RoboDK station: New Station (1).rdk

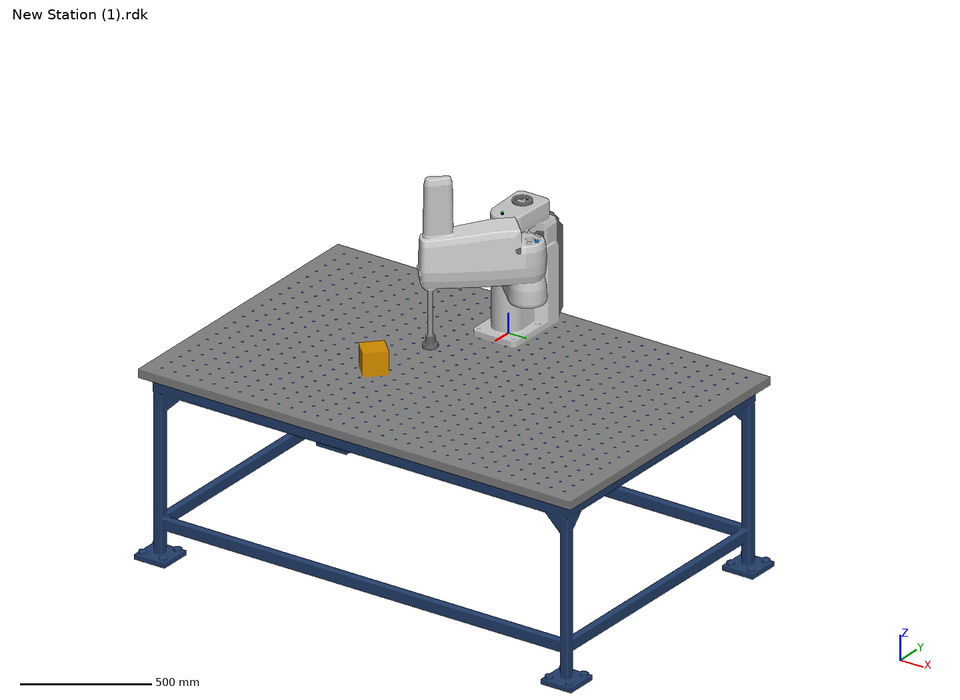
[picture v0: the station drawn from its stored meshes, robots at their saved joint values, targets as dots, program paths as lines]
Station New Station (1) (saved by RoboDK 5.3.2). Poses are relative to the parent item; angles as X-Y-Z fixed-axis rotations.
  - frame Adept Cobra s800 Base at (600, 400, 0) mm, rotated rx 0 ry 0 rz -90 deg
    - robot Adept Cobra s800: 4 axes, payload 2 kg, reach 800 mm, repeatability 0.018 mm, weight 43 kg
        modified DH rows (alpha deg, a mm, theta deg, d mm): 0, 0, 0, 0; 0, 425, 0, 0; 0, 375, 0, 184 linear; 180, 0, 0, 0
        joint limits [-105, -157.5, 0, -360] to [105, 157.5, 210, 360]; home [0, 0, 0, 0]; saved at [45, -90, 0, 0]
  - object Cube 100mm at (370, -230, 0) mm, rotated rx 0 ry 0 rz 45 deg, size 100 x 100 x 100 mm, geometry from Cube-100mm.sld
  - object SICK VSPP-5f2113 at (0, 0, 1400) mm, rotated rx 180 ry 0 rz -180 deg, size 53 x 116 x 38 mm, geometry from Cam2D_SICK_VSPP_5F2113.sld
  - object Table 2000x1200x800 at (0, 0, 0) mm, size 2020 x 1340 x 800 mm, geometry from Table-2000mmx1200mmx800mm.sld
